Staubli VAL3: encTrajPtCartesianAck.pgx

public program encTrajPtCartesianAck()
begin
  // encode 'prefix' and 'header'
  call encPrefixHeader(rosTrajPtCartesianAck.prefix, rosTrajPtCartesianAck.header)

  // encode 'sequence' variable of body message (data)
  toBinary(rosTrajPtCartesianAck.cartesianTrajPt.nSeq,1,"-4l",rosTrajPtCartesianAck.body.nData)

  // encodings of all other fields ignored to save CPU time, since values are all zeros
end
